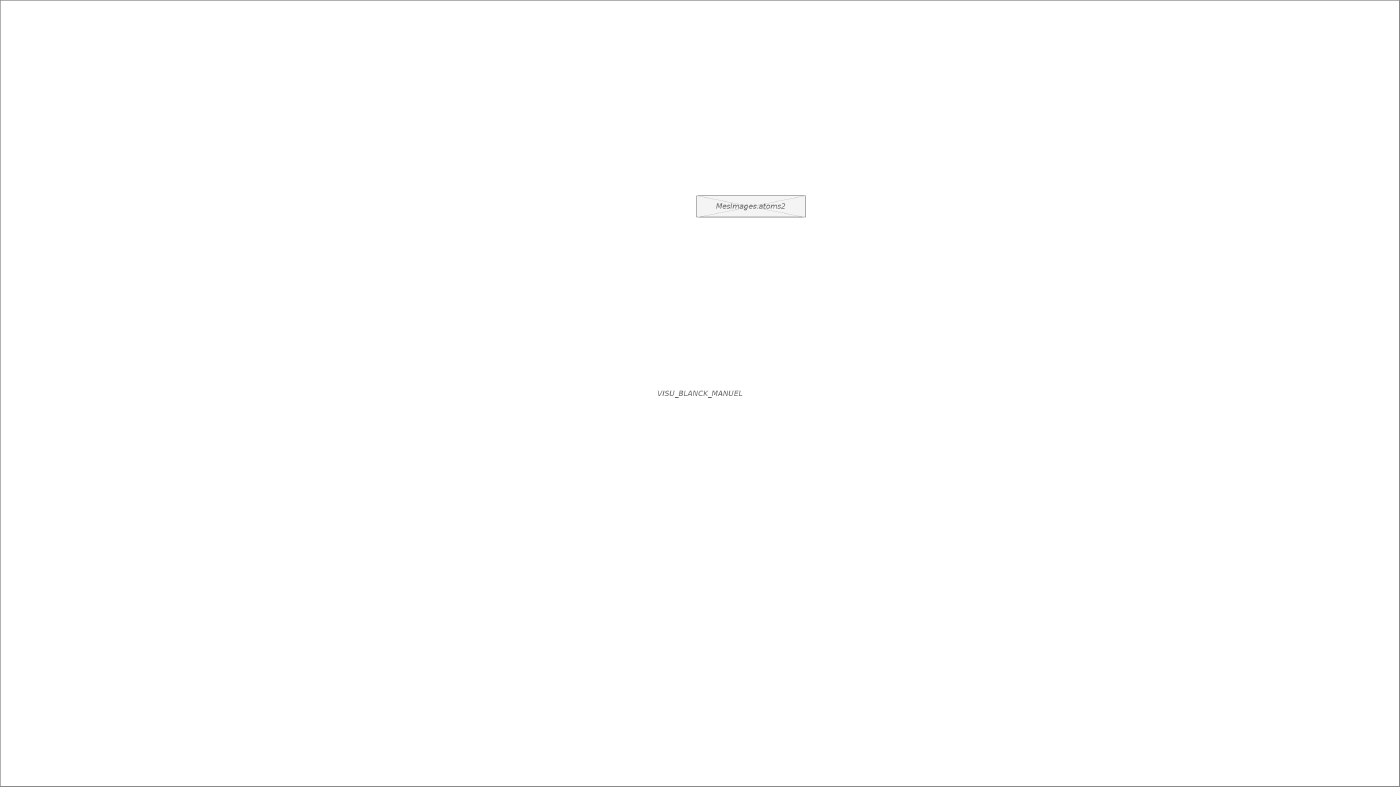
VISUALIZATION SYN_MANUEL  // 1920x1080, background image fond_blanc_1280_1024
    Frame (0,0 1920x1080), frame switch variable: VISU_INDEX_MANU
        shows VISU_BLANCK_MANUEL()
        shows VISU_XTAL6_ZOOM(m_Input_XTAL6 := .PRG_EVAP.QZ1)
        shows VISU_INFO(m_Input_CRYO := PRG_POMPAGE.COM_CRYOS, m_Input_PRG_POMPAGE := PRG_POMPAGE)
        shows VISU_VANNE_ASS_H_MANU(m_Input_Vanne := PRG_POMPAGE.POMPAGE.VS11, m_Input_State_Manu := MACHINE.STATE_Manu)
        [2]: m_Input_ID_NOM_XML=10, m_Input_INDEX_MOTEUR=2, m_Input_Ref_Trf=0
        p2655817705: .PRG_PUISSANCE.RF1
        p3040719188: .ENCEINTE.STATE_Manu
        p4051230613: PRG_MOUVEMENT_PS.ROTATION_PS
        p3521815518: PRG_MOUVEMENT_PS.TILT_PS
        p625233746: PRG_MOUVEMENT_PS.ROTATION_PS
    Image (955,268 150x30), image: MesImages.atoms2
END_VISUALIZATION

(* stored: Version 1.1.0.1, ProductVersion 3.1.4026.18
   Visu SYN_MANUEL: Id {cf29be52-0d29-455d-b3aa-628a3286359e} *)
